// TIA Portal V20 export
DATA_BLOCK "CS_Drive_PP"   // DB14, Motion_DB
// stored: InstanceOfName TO_SynchronousAxis, OfSystemLibElement TO_SynchronousAxis, OfSystemLibVersion 7.0
TO_SynchronousAxis   // technology object, version 7.0
// stored: Connection Interface Actor, InputAddress 9416, OutputAddress 9416
// stored: Connection Interface Sensor[1], InputAddress 9416, OutputAddress 9416, SensorIndexInActorTelegram 1
// stored: Connection Interface Torque, InputAddress 11360, OutputAddress 11360
// stored: SetPointCoupling Ref CS_Virtual_Axis, Type TO_PositioningAxis
// stored: SetPointCoupling Ref CS_Drive_PL, Type TO_SynchronousAxis
   // // inherited from TO_PositioningAxis
   // // inherited from TO_SpeedAxis
   // // inherited from TO_Axis
   // // inherited from TO_Object
   // VAR
   //    Actor : TO_Struct_Actor;
   //    LoadGear : TO_Struct_LoadGear;
   // END_VAR
   // VAR
   //    Sensor : Array[1..4] of TO_Struct_Sensor;
   //    Mechanics : TO_Struct_Mechanics;
   //    PositionControl : TO_Struct_PositionControl;
   //    DynamicAxisModel : TO_Struct_DynamicAxisModel;
   // END_VAR
   // VAR
   //    StatusSynchronizedMotion { ExternalWritable := 'False'; S7_SetPoint := 'True'} : TO_Struct_StatusSynchronizedMotion;
   // END_VAR
BEGIN
   Actor.InverseDirection := true;
   Actor.DataAdaption := 1;
   Actor.Interface.AddressIn.RID := 16#208072a;
   Actor.Interface.AddressIn.AREA := 16#81;
   Actor.Interface.AddressIn.OFFSET := 9416;
   Actor.Interface.AddressOut.RID := 16#208072b;
   Actor.Interface.AddressOut.AREA := 16#82;
   Actor.Interface.AddressOut.OFFSET := 9416;
   Actor.Interface.EnableTorqueData := true;
   Actor.Interface.TorqueDataAddressIn.RID := 16#2080742;
   Actor.Interface.TorqueDataAddressIn.AREA := 16#81;
   Actor.Interface.TorqueDataAddressIn.OFFSET := 11360;
   Actor.Interface.TorqueDataAddressOut.RID := 16#2080743;
   Actor.Interface.TorqueDataAddressOut.AREA := 16#82;
   Actor.Interface.TorqueDataAddressOut.OFFSET := 11360;
   Actor.DriveParameter.ReferenceSpeed := 6000.0;
   Actor.DriveParameter.MaxSpeed := 6000.0;
   Actor.DriveParameter.ReferenceTorque := 47.04;
   LoadGear.Numerator := 6843;
   LoadGear.Denominator := 100;
   Sensor[1]."Type" := 2;
   Sensor[1].InverseDirection := true;
   Sensor[1].DataAdaption := 1;
   Sensor[1].Interface.AddressIn.RID := 16#208072a;
   Sensor[1].Interface.AddressIn.AREA := 16#81;
   Sensor[1].Interface.AddressIn.OFFSET := 9416;
   Sensor[1].Interface.AddressOut.RID := 16#208072b;
   Sensor[1].Interface.AddressOut.AREA := 16#82;
   Sensor[1].Interface.AddressOut.OFFSET := 9416;
   Sensor[1].Parameter.FineResolutionXist2 := 0;
   Sensor[1].Parameter.DeterminableRevolutions := 4096;
   Mechanics.LeadScrew := 1256.0;
   PositionControl.Kv := 1.5;
   PositionControl.EnableDSC := true;
   DynamicAxisModel.VelocityTimeConstant := 0.004;
   Actor.Interface.EnableTorqueData := True;
   _Actor.Interface.Telegram := 105;
   _Actor.DataAdaptionOffline := True;
   _Sensor[1].Interface.Telegram := 105;
   _Sensor[1].DataAdaptionOffline := True;
END_DATA_BLOCK
